FUNCTION_BLOCK READ_Manufacturer_label
VAR_INPUT
	NodeID		: BYTE; (* This Port No. addresses the CANopen Node (see System Manager) *)	
	Start		: BOOL;
END_VAR
VAR_OUTPUT
	Label_Out	: ST_Manufacturer_label;
	Finished	: BOOL := FALSE;
END_VAR
VAR
	Index		: INT;
	Label		: ST_Manufacturer_label;
	SDO_READ 	: FB_SDO_READ;	
	SDO_READ_REAL 	: FB_SDO_READ_REAL;	
	SDO_WRITE 	: FB_SDO_WRITE;
	WriteData	: ARRAY [0..255] OF BYTE;		
	CAN_Objects	: INT;
END_VAR

// Restart after complete run
IF (Index = 255) AND Start THEN
	Index := 0;
END_IF


IF NOT (Index = 255) THEN 
	SDO_READ(StartReading:=FALSE);
	SDO_READ_REAL(StartReading:=FALSE);
END_IF
	
	
CASE Index OF	
	0: // Start reading Serial_Number
		IF Start THEN		
			Finished := FALSE;
			SDO_READ(	
				AdsNetID		:= GLB.ADSNetID_CAN,
				PortNr			:= 16#1000 + GLB.NodeID,
				CO_Index		:= 16#41C0,
				CO_SubIndex		:= 16#01,
				DataLength		:= 4,
				StartReading	:= TRUE	
			);	
			Index := Index + 1;
		END_IF
		
	1: // Serial_Number is read
		IF SDO_READ.ReadDataAvailable THEN
			Label.Serial_Number := SHL(BYTE_TO_DWORD(SDO_READ.ReadData[3]),24) + SHL(BYTE_TO_DWORD(SDO_READ.ReadData[2]),16) + SHL(BYTE_TO_DWORD(SDO_READ.ReadData[1]),8) + BYTE_TO_DWORD(SDO_READ.ReadData[0]);				
			Index := Index + 1;
		END_IF

	
	2: // Start reading Min_v
		SDO_READ(	
			AdsNetID		:= GLB.ADSNetID_CAN,
			PortNr			:= 16#1000 + GLB.NodeID,
			CO_Index		:= 16#41C0,
			CO_SubIndex		:= 16#03,
			DataLength		:= 4,
			StartReading	:= TRUE	
		);	
		Index := Index + 1;
	
	3: // Min_v is read
		IF SDO_READ.ReadDataAvailable THEN
			Label.Min_v := SHL(BYTE_TO_DWORD(SDO_READ.ReadData[3]),24) + SHL(BYTE_TO_DWORD(SDO_READ.ReadData[2]),16) + SHL(BYTE_TO_DWORD(SDO_READ.ReadData[1]),8) + BYTE_TO_DWORD(SDO_READ.ReadData[0]);				
			Index := Index + 1;
		END_IF
		
		
	4: // Start reading Max_v
		SDO_READ(	
			AdsNetID		:= GLB.ADSNetID_CAN,
			PortNr			:= 16#1000 + GLB.NodeID,
			CO_Index		:= 16#41C0,
			CO_SubIndex		:= 16#04,
			DataLength		:= 4,
			StartReading	:= TRUE	
		);	
		Index := Index + 1;
		
	5: // Max_v is read
		IF SDO_READ.ReadDataAvailable THEN
			Label.Max_v := SHL(BYTE_TO_DWORD(SDO_READ.ReadData[3]),24) + SHL(BYTE_TO_DWORD(SDO_READ.ReadData[2]),16) + SHL(BYTE_TO_DWORD(SDO_READ.ReadData[1]),8) + BYTE_TO_DWORD(SDO_READ.ReadData[0]);				
			Index := Index + 1;
		END_IF
		
		
	6: // Start reading Motor_rated_current
		SDO_READ(	
			AdsNetID		:= GLB.ADSNetID_CAN,
			PortNr			:= 16#1000 + GLB.NodeID,
			CO_Index		:= 16#41C0,
			CO_SubIndex		:= 16#05,
			DataLength		:= 4,
			StartReading	:= TRUE	
		);	
		Index := Index + 1;
		
	7: // Motor_rated_current is read
		IF SDO_READ.ReadDataAvailable THEN
			Label.Motor_rated_current := SHL(BYTE_TO_DWORD(SDO_READ.ReadData[3]),24) + SHL(BYTE_TO_DWORD(SDO_READ.ReadData[2]),16) + SHL(BYTE_TO_DWORD(SDO_READ.ReadData[1]),8) + BYTE_TO_DWORD(SDO_READ.ReadData[0]);				
			Index := Index + 1;
		END_IF
		
		
	8: // Start reading Drive_rated_current
		SDO_READ(	
			AdsNetID		:= GLB.ADSNetID_CAN,
			PortNr			:= 16#1000 + GLB.NodeID,
			CO_Index		:= 16#41C0,
			CO_SubIndex		:= 16#06,
			DataLength		:= 4,
			StartReading	:= TRUE	
		);	
		Index := Index + 1;
			
	9: // Drive_rated_current is read
		IF SDO_READ.ReadDataAvailable THEN
			Label.Drive_rated_current := SHL(BYTE_TO_DWORD(SDO_READ.ReadData[3]),24) + SHL(BYTE_TO_DWORD(SDO_READ.ReadData[2]),16) + SHL(BYTE_TO_DWORD(SDO_READ.ReadData[1]),8) + BYTE_TO_DWORD(SDO_READ.ReadData[0]);				
			Index := Index + 1;
		END_IF
		
		
	10: // Start reading Max_current
		SDO_READ(	
			AdsNetID		:= GLB.ADSNetID_CAN,
			PortNr			:= 16#1000 + GLB.NodeID,
			CO_Index		:= 16#41C0,
			CO_SubIndex		:= 16#07,
			DataLength		:= 4,
			StartReading	:= TRUE	
		);	
		Index := Index + 1;

	11: // Max_current is read
		IF SDO_READ.ReadDataAvailable THEN
			Label.Max_current := SHL(BYTE_TO_WORD(SDO_READ.ReadData[1]),8) + BYTE_TO_WORD(SDO_READ.ReadData[0]);				
			Index := Index + 1;
		END_IF
		
		
	12: // Start reading Motor_rated_torque
		SDO_READ(	
			AdsNetID		:= GLB.ADSNetID_CAN,
			PortNr			:= 16#1000 + GLB.NodeID,
			CO_Index		:= 16#41C0,
			CO_SubIndex		:= 16#08,
			DataLength		:= 4,
			StartReading	:= TRUE	
		);	
		Index := Index + 1;
	
	13: // Motor_rated_torque is read
		IF SDO_READ.ReadDataAvailable THEN
			Label.Motor_rated_torque := SHL(BYTE_TO_DWORD(SDO_READ.ReadData[3]),24) + SHL(BYTE_TO_DWORD(SDO_READ.ReadData[2]),16) + SHL(BYTE_TO_DWORD(SDO_READ.ReadData[1]),8) + BYTE_TO_DWORD(SDO_READ.ReadData[0]);				
			Index := Index + 1;
		END_IF			
		
		
	14: // Start reading Max_torque
		SDO_READ(	
			AdsNetID		:= GLB.ADSNetID_CAN,
			PortNr			:= 16#1000 + GLB.NodeID,
			CO_Index		:= 16#41C0,
			CO_SubIndex		:= 16#09,
			DataLength		:= 2,
			StartReading	:= TRUE	
		);	
		Index := Index + 1;		
		
	15: // Max_torque is read
		IF SDO_READ.ReadDataAvailable THEN
			Label.Max_torque := SHL(BYTE_TO_WORD(SDO_READ.ReadData[1]),8) + BYTE_TO_WORD(SDO_READ.ReadData[0]);
			Index := Index + 1;
		END_IF
		
		
	16: // Start reading Motor_rated_speed
		SDO_READ(	
			AdsNetID		:= GLB.ADSNetID_CAN,
			PortNr			:= 16#1000 + GLB.NodeID,
			CO_Index		:= 16#41C0,
			CO_SubIndex		:= 16#0A,
			DataLength		:= 4,
			StartReading	:= TRUE	
		);	
		Index := Index + 1;
			
	17: // Motor_rated_speed is read
		IF SDO_READ.ReadDataAvailable THEN
			Label.Motor_rated_speed := SHL(BYTE_TO_DWORD(SDO_READ.ReadData[3]),24) + SHL(BYTE_TO_DWORD(SDO_READ.ReadData[2]),16) + SHL(BYTE_TO_DWORD(SDO_READ.ReadData[1]),8) + BYTE_TO_DWORD(SDO_READ.ReadData[0]);				
			Index := Index + 1;
		END_IF
		
		
	18: // Start reading Number_of_pole_pairs
		SDO_READ(	
			AdsNetID		:= GLB.ADSNetID_CAN,
			PortNr			:= 16#1000 + GLB.NodeID,
			CO_Index		:= 16#41C0,
			CO_SubIndex		:= 16#0B,
			DataLength		:= 2,
			StartReading	:= TRUE	
		);	
		Index := Index + 1;			
		
	19: // Reading Number_of_pole_pairs, next reading Motor_torque_constant
		IF SDO_READ.ReadDataAvailable THEN
			Label.Number_of_pole_pairs := SHL(BYTE_TO_WORD(SDO_READ.ReadData[1]),8) + BYTE_TO_WORD(SDO_READ.ReadData[0]);
			Index := Index + 1;
		END_IF
		
		
	20: // Start reading Motor_torque_constant
		SDO_READ_REAL(	
				AdsNetID		:= GLB.ADSNetID_CAN,
				PortNr			:= 16#1000 + GLB.NodeID,
				CO_Index		:= 16#41C0,
				CO_SubIndex		:= 16#0C,
				StartReading	:= TRUE	
			);	
			Index := Index + 1;			
		
	21: // Motor_torque_constant is read
		IF SDO_READ_REAL.ReadDataAvailable THEN
			Label.Motor_torque_constant := SDO_READ_REAL.ReadData;
			Index := Index + 1;
		END_IF
		
		
	22: // Start reading Flux_producing_P_gain
		SDO_READ_REAL(	
			AdsNetID		:= GLB.ADSNetID_CAN,
			PortNr			:= 16#1000 + GLB.NodeID,
			CO_Index		:= 16#41C0,
			CO_SubIndex		:= 16#0D,
			StartReading	:= TRUE	
		);	
		Index := Index + 1;
					
	23: // Flux_producing_P_gain is read
		IF SDO_READ_REAL.ReadDataAvailable THEN
			Label.Flux_producing_P_gain := SDO_READ_REAL.ReadData;
			Index := Index + 1;
		END_IF
		
		
	24: // Start reading Flux_producing_I_gain
		SDO_READ_REAL(	
			AdsNetID		:= GLB.ADSNetID_CAN,
			PortNr			:= 16#1000 + GLB.NodeID,
			CO_Index		:= 16#41C0,
			CO_SubIndex		:= 16#0E,
			StartReading	:= TRUE	
		);	
		Index := Index + 1;

	25: // Flux_producing_I_gain is read
		IF SDO_READ_REAL.ReadDataAvailable THEN
			Label.Flux_producing_I_gain := SDO_READ_REAL.ReadData;
			Index := Index + 1;
		END_IF
		
		
	26: // Start reading Torque_producing_P_gain
		SDO_READ_REAL(	
			AdsNetID		:= GLB.ADSNetID_CAN,
			PortNr			:= 16#1000 + GLB.NodeID,
			CO_Index		:= 16#41C0,
			CO_SubIndex		:= 16#0F,
			StartReading	:= TRUE	
		);	
		Index := Index + 1;
		
	27: // Torque_producing_P_gain is read
		IF SDO_READ_REAL.ReadDataAvailable THEN
			Label.Torque_producing_P_gain := SDO_READ_REAL.ReadData;
			Index := Index + 1;
		END_IF
		
		
	28: // Start reading Torque_producing_I_gain
		SDO_READ_REAL(	
			AdsNetID		:= GLB.ADSNetID_CAN,
			PortNr			:= 16#1000 + GLB.NodeID,
			CO_Index		:= 16#41C0,
			CO_SubIndex		:= 16#10,
			StartReading	:= TRUE	
		);	
		Index := Index + 1;

	29: // Torque_producing_I_gain is read
		IF SDO_READ_REAL.ReadDataAvailable THEN
			Label.Torque_producing_I_gain := SDO_READ_REAL.ReadData;
			Index := Index + 1;
		END_IF
		
		
	30: // Start reading Magnetic_encoder_offset
		SDO_READ(	
			AdsNetID		:= GLB.ADSNetID_CAN,
			PortNr			:= 16#1000 + GLB.NodeID,
			CO_Index		:= 16#41C0,
			CO_SubIndex		:= 16#11,
			DataLength		:= 2,
			StartReading	:= TRUE	
		);	
		Index := Index + 1;

	31: // Magnetic_encoder_offset is read
		IF SDO_READ.ReadDataAvailable THEN
			Label.Magnetic_encoder_offset := SHL(BYTE_TO_WORD(SDO_READ.ReadData[1]),8) + BYTE_TO_WORD(SDO_READ.ReadData[0]);				
			Index := Index + 1;
		END_IF
		
		
	32: // Start reading Motor_with_brake
		SDO_READ(	
			AdsNetID		:= GLB.ADSNetID_CAN,
			PortNr			:= 16#1000 + GLB.NodeID,
			CO_Index		:= 16#41C0,
			CO_SubIndex		:= 16#12,
			DataLength		:= 2,
			StartReading	:= TRUE	
		);	
		Index := Index + 1;

	33: // Motor_with_brake is read
		IF SDO_READ.ReadDataAvailable THEN
			Label.Motor_with_brake := SHL(BYTE_TO_WORD(SDO_READ.ReadData[1]),8) + BYTE_TO_WORD(SDO_READ.ReadData[0]);				
			Index := Index + 1;
		END_IF
		
		
	34: // Start reading Encoder_mode_adjust
		SDO_READ(	
			AdsNetID		:= GLB.ADSNetID_CAN,
			PortNr			:= 16#1000 + GLB.NodeID,
			CO_Index		:= 16#41C0,
			CO_SubIndex		:= 16#13,
			DataLength		:= 2,
			StartReading	:= TRUE	
		);	
		Index := Index + 1;

	35: // Encoder_mode_adjust is read
		IF SDO_READ.ReadDataAvailable THEN
			Label.Encoder_mode_adjust := SHL(BYTE_TO_WORD(SDO_READ.ReadData[1]),8) + BYTE_TO_WORD(SDO_READ.ReadData[0]);				
			Index := Index + 1;
		END_IF
		
		
	36: // Start reading Motor_max_speed
		SDO_READ(	
			AdsNetID		:= GLB.ADSNetID_CAN,
			PortNr			:= 16#1000 + GLB.NodeID,
			CO_Index		:= 16#41C0,
			CO_SubIndex		:= 16#14,
			DataLength		:= 2,
			StartReading	:= TRUE	
		);	
		Index := Index + 1;
					
	37: // Motor_max_speed is read
		IF SDO_READ.ReadDataAvailable THEN
			Label.Motor_max_speed := SHL(BYTE_TO_WORD(SDO_READ.ReadData[1]),8) + BYTE_TO_WORD(SDO_READ.ReadData[0]);				
			Index := Index + 1;
		END_IF
				
		
	38: // Start reading Rotor_inertia
		SDO_READ_REAL(	
			AdsNetID		:= GLB.ADSNetID_CAN,
			PortNr			:= 16#1000 + GLB.NodeID,
			CO_Index		:= 16#41C0,
			CO_SubIndex		:= 16#15,
			StartReading	:= TRUE	
		);	
		Index := Index + 1;
					
	39: // Rotor_inertia is read
		IF SDO_READ_REAL.ReadDataAvailable THEN
			Label.Rotor_inertia := SDO_READ_REAL.ReadData;
			Index := Index + 1;
		END_IF
		
		
	40: // Start reading Motor_time_at_peak
		SDO_READ_REAL(	
			AdsNetID		:= GLB.ADSNetID_CAN,
			PortNr			:= 16#1000 + GLB.NodeID,
			CO_Index		:= 16#41C0,
			CO_SubIndex		:= 16#17,
			StartReading	:= TRUE	
		);	
		Index := Index + 1;
					
	41: // Motor_time_at_peak is read
		IF SDO_READ_REAL.ReadDataAvailable THEN
			Label.Motor_time_at_peak := SDO_READ_REAL.ReadData;
			Index := Index + 1;
		END_IF
		
		
	42: // Start reading Drive_time_at_peak
		SDO_READ_REAL(	
			AdsNetID		:= GLB.ADSNetID_CAN,
			PortNr			:= 16#1000 + GLB.NodeID,
			CO_Index		:= 16#41C0,
			CO_SubIndex		:= 16#18,
			StartReading	:= TRUE	
		);	
		Index := Index + 1;
		
	43: // Drive_time_at_peak is read
		IF SDO_READ_REAL.ReadDataAvailable THEN
			Label.Drive_time_at_peak := SDO_READ_REAL.ReadData;
			Index := Index + 1;
		END_IF
		
		
	44: // Start reading Singleturn_resolution
		SDO_READ(	
			AdsNetID		:= GLB.ADSNetID_CAN,
			PortNr			:= 16#1000 + GLB.NodeID,
			CO_Index		:= 16#41C0,
			CO_SubIndex		:= 16#19,
			DataLength		:= 1,
			StartReading	:= TRUE	
		);	
		Index := Index + 1;
					
	45: // Singleturn_resolution is read 
		IF SDO_READ.ReadDataAvailable THEN
			Label.Singleturn_resolution := SDO_READ.ReadData[0];				
			Index := Index + 1;
		END_IF		
		
		
	46: // Start reading Multiturn_resolution
		SDO_READ(	
			AdsNetID		:= GLB.ADSNetID_CAN,
			PortNr			:= 16#1000 + GLB.NodeID,
			CO_Index		:= 16#41C0,
			CO_SubIndex		:= 16#1A,
			DataLength		:= 1,
			StartReading	:= TRUE	
		);	
		Index := Index + 1;
			
	47: // Multiturn_resolution is read
		IF SDO_READ.ReadDataAvailable THEN
			Label.Multiturn_resolution := SDO_READ.ReadData[0];	
			Index := 255;
		END_IF		
				
		
	255: // Finished 
		Label_Out := Label;
		Finished := TRUE;
				
		
	ELSE
		Index := 255;
			
END_CASE

END_FUNCTION_BLOCK

(* stored: Version 1.1.0.1, ProductVersion 3.1.4024.11
   POU READ_Manufacturer_label: Id {15d1b11f-1b71-4f19-97bd-14c8867b098b}, SpecialFunc None *)
